// TwinCAT 3 PLC project MicroTestStandPPM
// ProgramVersion: 3.1.4020.5
// libraries:
//   lcls-twincat-motion, * (SLAC)
//   lcls2-cc-lib, * (SLAC)
//   Tc2_Standard, * (Beckhoff Automation GmbH)
//   Tc2_System, * (Beckhoff Automation GmbH)
//   Tc2_Utilities, * (Beckhoff Automation GmbH)
//   Tc3_Module, * (Beckhoff Automation GmbH)
//   VisuDialogs
//   VisuSymbols,3.5.10.0,System
// project tree:
//   DUTs/ DUT_MotionStage_Extras.TcDUT (not stored)
//   / GlobalTextList.TcGTLO (not stored), PlcTask.TcTTO (not stored), VISU_TASK.TcTTO (not stored)
//   POUs/ Main.TcPOU
//   VISUs/ Visualization.TcVIS (not stored), VisualizationManager.TcVMO (not stored), VISU_MotionStage.TcVIS (not stored)
// real-time tasks:
//   TASK PlcTask: cycle T#1ms, priority 20, ADS port 350
//   TASK VISU_TASK: cycle T#200000us, priority 30, ADS port 351
// motion (NC):
// I/O:
//   DEVICE Device 1 (EtherCAT), AmsNetId 172.21.148.185.2.1
//     EK1200
//     EK1100 [EK1100 EtherCAT Coupler (2A E-Bus)]
//       EL7041
//       EL2004 [EL2004 4Ch. Dig. Output 24V, 0.5A]
//       EL5042 [EL5042 2Ch. BiSS-C Encoder]
//       EL9011
// variable links:
//   MicroTestStandPPM Instance <-> Device 1 (EtherCAT)/EK1100/EL2004
//     PlcTask Outputs/Main.M1.bBrakeRelease <-> Channel 1/Output
//   MicroTestStandPPM Instance <-> Device 1 (EtherCAT)/EK1100/EL5042
//     PlcTask Inputs/Main.iRawEncoder <-> FB Inputs Channel 1/Position
//   MicroTestStandPPM Instance <-> Device 1 (EtherCAT)/EK1100/EL7041
//     PlcTask Inputs/Main.M1.bLimitBackwardEnable <-> STM Status/Status/Digital input 2
//     PlcTask Inputs/Main.M1.bLimitForwardEnable <-> STM Status/Status/Digital input 1
//   MicroTestStandPPM Instance <-> NC-Task 1 SAF/Axes/MMS_Y
//     PlcTask Inputs/Main.M1.Axis.NcToPlc <-> Outputs/ToPlc
//     PlcTask Outputs/Main.M1.Axis.PlcToNc <-> Inputs/FromPlc

// ---- POUs/Main.TcPOU
PROGRAM Main
VAR
	{attribute 'pytmc' := '
        pv: TST:PPM:MMS:01
		io: io
	'}
	{attribute 'TcLinkTo' := '.bLimitForwardEnable  := TIIB[EL7041]^STM Status^Status^Digital input 1;
	                          .bLimitBackwardEnable := TIIB[EL7041]^STM Status^Status^Digital input 2;
	                          .bBrakeRelease        := TIIB[EL2004]^Channel 1^Output'}
	M1: DUT_MotionStage;
	M1_Extras: DUT_MotionStage_Extras;
	
	{attribute 'pytmc' := '
		pv: TST:PPM
		io: io
	'}
    (*
	{attribute 'TcLinkTo' := '.fbGige.iIlluminatorINT := TIIB[EL4004]^AO Outputs Channel 1^Analog output;
	                          .fbGige.bGigePower := TIIB[EL2004]^Channel 2^Output;
							  .fbPowerMeter.iVoltageINT := TIIB[EL3062]^AI Standard Channel 1^Value;
							  .fbPowerMeter.fbThermoCouple.bError := TIIB[EL3314]^TC Inputs Channel 1^Status^Error;
							  .fbPowerMeter.fbThermoCouple.bUnderrange := TIIB[EL3314]^TC Inputs Channel 1^Status^Underrange;
							  .fbPowerMeter.fbThermoCouple.bOverrange := TIIB[EL3314]^TC Inputs Channel 1^Status^Overrange;
							  .fbPowerMeter.fbThermoCouple.iRaw := TIIB[EL3314]^TC Inputs Channel 1^Value;
							  .fbYagThermoCouple.bError := TIIB[EL3314]^TC Inputs Channel 2^Status^Error;
							  .fbYagThermoCouple.bUnderrange := TIIB[EL3314]^TC Inputs Channel 2^Status^Underrange;
							  .fbYagThermoCouple.bOverrange := TIIB[EL3314]^TC Inputs Channel 2^Status^Overrange;
							  .fbYagThermoCouple.iRaw := TIIB[EL3314]^TC Inputs Channel 2^Value'}
                              *)
	fbPPM: FB_PPM;
	
	{attribute 'pytmc' := '
		pv: TST:PPM:MMS:01:ENC_RAW
		io: i
	'}
	iAdjustedEncoder: UDINT;
	iRawEncoder AT %I*: ULINT;
	iMaxLINT: ULINT := 18446744073709551615;
	
	bStartup: BOOL := TRUE;
END_VAR

fbPPM(stYStage := M1);
M1.bHardwareEnable := TRUE;
iAdjustedEncoder :=  ULINT_TO_UDINT(iMaxLINT - iRawEncoder);

M1_Extras.bVisuHighLim := NOT M1.bAllForwardEnable;
M1_Extras.bVisuLowLim := NOT M1.bAllBackwardEnable;

IF bStartup THEN
	bStartup := FALSE;
	M1.fVelocity := 1;
	M1.fAcceleration := 200;
	M1.fDeceleration := 200;
END_IF

END_PROGRAM
